// TIA Portal V18 export
// export: Created 2026-03-12T16:04:34.6914029Z, ExportSetting WithDefaults, DisplayName Totally Integrated Automation Portal, DisplayVersion V18 Update 5, DisplayName TIA Portal Openness, DisplayVersion V18 Update 5, DisplayName TIA Portal Version Control Interface, DisplayVersion V18, DisplayName SINAMICS Startdrive Advanced, DisplayVersion V18, DisplayName SINAMICS Startdrive G130, G150, S120, S150, SINAMICS MV, S210, DisplayVersion V18, DisplayName SINAMICS Startdrive G110M, G120, G120C, G120D, G120P, G115D, DisplayVersion V18, DisplayName STEP 7 Professional, DisplayVersion V18 Update 5, DisplayName STEP 7 Safety, DisplayVersion V18, DisplayName WinCC Professional, DisplayVersion V18 Update 5
FUNCTION_BLOCK "FB_LIGA/DESLIGA MODO AUTO"   // FB8, LAD
TITLE = Function Block LIGA/DESLIGA MODO AUTO
{ S7_Optimized_Access := 'TRUE' }
VERSION : 0.1
// Bloco para alternância dinâmica do tempo para ligar e desligar bomba.
// Network 1: Atribuição do sinal de liga
// Network 2: Function Block CONTADOR: Contador de tempo para bomba ligada
// Network 3: Comparativo de bomba ligada com tempo cadastrado para ficar ligada
// Network 4: Function Block CONTADOR: Contador de tempo para bomba desligada
// Network 5: Comparativo de bomba desligada com tempo cadastrado para ficar desligada
// Network 6: Transferindo sinal de bomba ligada/desligada para fora do bloco
// stored: AutoNumber true, IsIECCheckEnabled false, IsRetainMemResEnabled false, MemoryReserve 100, SetENOAutomatically false, UDAEnableTagReadback false
   VAR_INPUT
      REMOTO_AUTO : Bool;   // Modo Remoto Automático
      CAD_TEMPO_LIGADA : Real;   // Cadastro tempo para bomba ficar ligada
      CAD_TEMPO_DESLIGADA : Real;   // Cadastro tempo para bomba ficar desligada
      TEMPO_ALTERNANCIA : Bool;   // Controle de alternancia entre bombas
   END_VAR
   VAR_OUTPUT
      HABILITA_LIGA_AUTO : Bool;   // Habilita Liga em Modo Automático
   END_VAR
   VAR_IN_OUT
      TEMPO_LIGADA_AUTO_SEG : Real;   // Tempo de bomba ligada em Modo Automático (segundos)
      TEMPO_LIGADA_AUTO_MIN : Real;   // Tempo de bomba ligada em Modo Automático (minutos)
      TEMPO_LIGADA_AUTO_HOR : Real;   // Tempo de bomba ligada em Modo Automático (horas)
      TEMPO_DESLIGADA_AUTO_SEG : Real;   // Tempo de bomba desligada em Modo Automático (segundos)
      TEMPO_DESLIGADA_AUTO_MIN : Real;   // Tempo de bomba desligada em Modo Automático (minutos)
      TEMPO_DESLIGADA_AUTO_HOR : Real;   // Tempo de bomba desligada em Modo Automático (horas)
   END_VAR
   VAR
      DESLIGA_AUTO : Bool;   // Desliga bomba em Modo Automático
      LIGA_AUTO : Bool;   // Liga bomba em Modo Automático
      MINUTEIRO_LIGADA : "FB CONTADOR";
      MINUTEIRO_DESLIGADA : "FB CONTADOR";
      TEMPO_LIGADA_AUTO_HORA : Bool;   // Tempo de bomba desligada em Modo Automático (em horas)
   END_VAR
BEGIN

REGION Network 1: Atribuição do sinal de liga
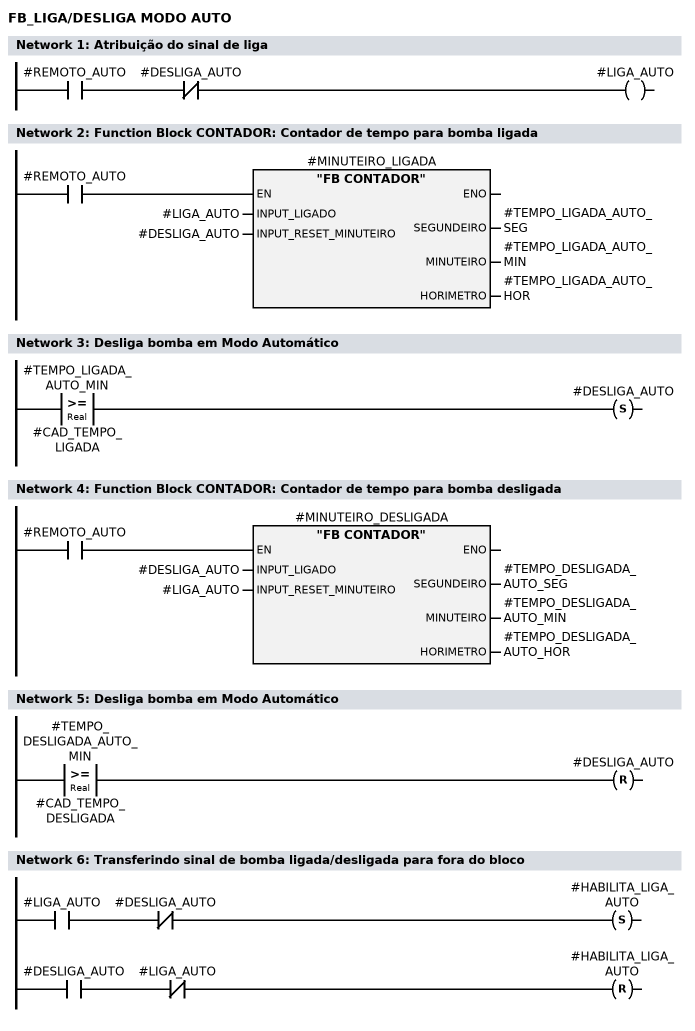
   RUNG wire#powerrail
      Contact( #REMOTO_AUTO )
      I_Contact( #DESLIGA_AUTO )
      Coil( #LIGA_AUTO )
   END_RUNG
   // the same network as SCL:
   #LIGA_AUTO := #REMOTO_AUTO AND NOT #DESLIGA_AUTO;
END_REGION

REGION Network 2: Function Block CONTADOR: Contador de tempo para bomba ligada
   RUNG wire#powerrail
      Contact( #REMOTO_AUTO )
      #MINUTEIRO_LIGADA(INPUT_LIGADO := #LIGA_AUTO, INPUT_RESET_MINUTEIRO := #DESLIGA_AUTO, SEGUNDEIRO => #TEMPO_LIGADA_AUTO_SEG, MINUTEIRO => #TEMPO_LIGADA_AUTO_MIN, HORIMETRO => #TEMPO_LIGADA_AUTO_HOR)
   END_RUNG
   // the same network as SCL:
   IF #REMOTO_AUTO THEN
       #MINUTEIRO_LIGADA(INPUT_LIGADO := #LIGA_AUTO,   // "FB CONTADOR"
                         INPUT_RESET_MINUTEIRO := #DESLIGA_AUTO,
                         SEGUNDEIRO => #TEMPO_LIGADA_AUTO_SEG,
                         MINUTEIRO => #TEMPO_LIGADA_AUTO_MIN,
                         HORIMETRO => #TEMPO_LIGADA_AUTO_HOR);
   END_IF;
END_REGION

REGION Network 3: Desliga bomba em Modo Automático
   RUNG wire#powerrail
      { S7_Templates := "SrcType := Real" } GE_Contact(in1 := #TEMPO_LIGADA_AUTO_MIN, in2 := #CAD_TEMPO_LIGADA)
      S_Coil( #DESLIGA_AUTO )
   END_RUNG
   // the same network as SCL:
   IF #TEMPO_LIGADA_AUTO_MIN >= #CAD_TEMPO_LIGADA THEN #DESLIGA_AUTO := TRUE; END_IF;
END_REGION

REGION Network 4: Function Block CONTADOR: Contador de tempo para bomba desligada
   RUNG wire#powerrail
      Contact( #REMOTO_AUTO )
      #MINUTEIRO_DESLIGADA(INPUT_LIGADO := #DESLIGA_AUTO, INPUT_RESET_MINUTEIRO := #LIGA_AUTO, SEGUNDEIRO => #TEMPO_DESLIGADA_AUTO_SEG, MINUTEIRO => #TEMPO_DESLIGADA_AUTO_MIN, HORIMETRO => #TEMPO_DESLIGADA_AUTO_HOR)
   END_RUNG
   // the same network as SCL:
   IF #REMOTO_AUTO THEN
       #MINUTEIRO_DESLIGADA(INPUT_LIGADO := #DESLIGA_AUTO,   // "FB CONTADOR"
                            INPUT_RESET_MINUTEIRO := #LIGA_AUTO,
                            SEGUNDEIRO => #TEMPO_DESLIGADA_AUTO_SEG,
                            MINUTEIRO => #TEMPO_DESLIGADA_AUTO_MIN,
                            HORIMETRO => #TEMPO_DESLIGADA_AUTO_HOR);
   END_IF;
END_REGION

REGION Network 5: Desliga bomba em Modo Automático
   RUNG wire#powerrail
      { S7_Templates := "SrcType := Real" } GE_Contact(in1 := #TEMPO_DESLIGADA_AUTO_MIN, in2 := #CAD_TEMPO_DESLIGADA)
      R_Coil( #DESLIGA_AUTO )
   END_RUNG
   // the same network as SCL:
   IF #TEMPO_DESLIGADA_AUTO_MIN >= #CAD_TEMPO_DESLIGADA THEN #DESLIGA_AUTO := FALSE; END_IF;
END_REGION

REGION Network 6: Transferindo sinal de bomba ligada/desligada para fora do bloco
   RUNG wire#powerrail
      Contact( #LIGA_AUTO )
      I_Contact( #DESLIGA_AUTO )
      S_Coil( #HABILITA_LIGA_AUTO )
   END_RUNG
   RUNG wire#powerrail
      Contact( #DESLIGA_AUTO )
      I_Contact( #LIGA_AUTO )
      R_Coil( #HABILITA_LIGA_AUTO )
   END_RUNG
   // the same network as SCL:
   IF #LIGA_AUTO AND NOT #DESLIGA_AUTO THEN #HABILITA_LIGA_AUTO := TRUE; END_IF;
   IF #DESLIGA_AUTO AND NOT #LIGA_AUTO THEN #HABILITA_LIGA_AUTO := FALSE; END_IF;
END_REGION
END_FUNCTION_BLOCK
